_CFC_ (* Continuous Function Chart, elements in execution order *)
#0 <>(SCHU_P2_2_M_MAXSPEED_PE, 0)
#1 AND(SCHU_P2_2_PE_PID_VKL, #0)
#2 Zad_PE:TON(IN: #1, PT: T#2s)
#3 SEL(#2.Q, SCHU_P2_2_M_MAXSPEED_CH, SCHU_P2_2_M_MAXSPEED_PE)
#4 SCHU_P2_2_M_MAXSPEED <= #3
#5 MOVE(EN: NOT #37.Q1, SCHU_P2_2_M_MAXSPEED)
#6 SCHU_P2_2_SPEEDMOTOR <= #5
#7 OR(M1_PUSK, M2_PUSK)
#8 AND(SCHU_P2_2_YA2_M_UST_VKL_UVEL_CHAST, SCHU_P2_2_UE1_TE_NM_UST)
#9 AND(SCHU_P2_2_YA3_M_UST_VKL_UVEL_CHAST, SCHU_P2_2_UE1_TE_NB_UST)
#10 AND(SCHU_P2_2_YA4_M_UST_VKL_UVEL_CHAST, SCHU_P2_2_UE3_TE_B_UST)
#11 AND(#8, #9, #10)
#12 OR(SCHU_P2_2_UE1_TE_M_UST, SCHU_P2_2_UE1_TE_B_UST, SCHU_P2_2_UE3_TE_M_UST, SCHU_P2_2_UST_RE_STOP)
#13 AND(SCHU_P2_2_YA2_B_UST_VKL_STER_REG, SCHU_P2_2_UE1_TE_M_UST)
#14 AND(SCHU_P2_2_UE1_TE_B_UST, SCHU_P2_2_YA3_B_UST_VKL_STER_REG)
#15 AND(SCHU_P2_2_YA4_B_UST_VKL_STER_REG, SCHU_P2_2_UE3_TE_M_UST)
#16 OR(#13, #14, #15)
#17 OR(SCHU_P2_2_M2_OBRBSM, SCHU_P2_2_M1_OBRBSM)
#18 AND(SCHU_P2_2_UST_RE_RABOTA, SCHU_P2_2_AVR_M)
#19 AND(NOT SCHU_P2_2_SA8_DI4_M, SCHU_P2_2_SA1_DI6_M)
#20 OR(SCHU_P2_2_SA1_DO1, SCHU_P2_2_SA8_DO8)
#21 AND(#17, #20)
#22 AND(#11, #21)
#23 SR_START_POV_REG:RS(SET: #22, RESET1: #12)
#24 AND(#16, #21)
#25 AND(#7, #20)
#26 OR(#18, #25)
#27 SEL(#23.Q1, SCHU_P2_2_SPEEDMOTOR, SCHU_P2_2_M_MAXSPEED)
#28 AND(SCHU_P2_2_YA4_M_UST_VKL_STER_REG, SCHU_P2_2_UE3_TE_B_UST)
#29 AND(#23.Q1, #25)
#30 SEL(#29, SCHU_P2_2_M_USKORENIE_PUSK, SCHU_P2_2_M_USKORENIE_UPR)
#31 AND(SCHU_P2_2_UE2_TE_NB_UST, SCHU_P2_2_YA3_M_UST_VKL_STER_REG)
#32 AND(SCHU_P2_2_SA8_DI4_M, NOT SCHU_P2_2_SA1_DI6_M)
#33 AND(SCHU_P2_2_YA2_M_UST_VKL_STER_REG, SCHU_P2_2_UE1_TE_NM_UST)
#34 SEL(SCHU_P2_2_UST_ZIMA, #31, #33)
#35 AND(#28, #34)
#36 OR(SCHU_P2_2_UST_RE_STOP, #35)
#37 SR_START_STER_REG:SR(SET1: #24, RESET: #36)
#38 AND(SCHU_P2_2_M_SB2_STER_REG, NOT #37.Q1)
#39 MOVE(EN: #38, SCHU_P2_2_M_MAXSPEED)
#40 SCHU_P2_2_SPEEDMOTOR <= #39
#41 OR(#23.Q1, #37.Q1)
#42 SEL(#37.Q1, #27, SCHU_P2_2_M_MINSPEED)
#43 SEL(#26, 0, #42)
#44 AND(#25, #37.Q1)
#45 SEL(#44, SCHU_P2_2_M_ZAMEDLENIE_OST, SCHU_P2_2_M_ZAMEDLENIE_UPR)
#46 SEL(SCHU_P2_2_UST_SET_STOP, #45, 1000)
#47 RR:RAMP_REAL(#43, #30, #46, T#1s, -)
#48 MOVE(EN: #41, #47)
#49 SCHU_P2_2_SPEEDMOTOR <= #48
#50 MOVE(EN: SCHU_P2_2_SA1_DO1, #47)
#51 SEL(#50.ENO, 0, #50)
#52 SEL(#19, #51, SCHU_P2_2_M_ZAD_RUCH)
#53 SCHU_P2_2_M1_ZAD_VN <= #52
#54 MOVE(EN: SCHU_P2_2_SA8_DO8, #47)
#55 SEL(#54.ENO, 0, #54)
#56 SEL(#32, #55, SCHU_P2_2_M_ZAD_RUCH)
#57 SCHU_P2_2_M2_ZAD_VN <= #56
#58 RT_KOMVKL_1:R_TRIG(CLK: SCHU_P2_2_UST_RE_PUSK)
#59 MOVE(EN: #58.Q, SCHU_P2_2_M_MAXSPEED)
#60 SCHU_P2_2_SPEEDMOTOR <= #59
#61 RT_KOMVKL_2:R_TRIG(CLK: TRUE)
#62 MOVE(EN: #61.Q, 5)
#63 SCHU_P2_2_M_ZAD_RUCH <= #62
_END_CFC_
END_PROGRAM

(* POU IM/P1_Upr, CFC *)
PROGRAM P1_Upr
VAR
	fb_HVACMS_P1: FB_HVACMotor1Speed;
	SR_P1: SR;
	startDelay_P1: TIME := T#0s;
	stopDelay_P1: TIME := T#0s;
	delayFBC_P1: TIME;
	feedbPT_P1: TIME :=T#10s ;
	delayFBP_P1: TIME := T#10s;
	TON_P1_OTKL_Leto: TON;
	TON_P1_VKL_Leto: TON;
END_VAR
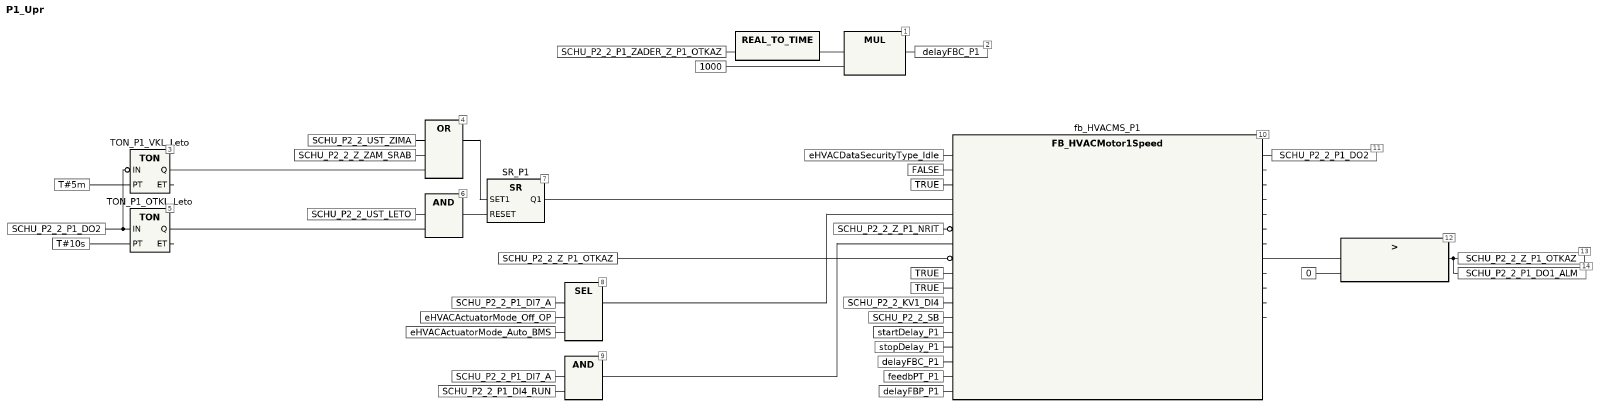
_CFC_ (* Continuous Function Chart, elements in execution order *)
#0 REAL_TO_TIME(SCHU_P2_2_P1_ZADER_Z_P1_OTKAZ)
#1 MUL(#0, 1000)
#2 delayFBC_P1 <= #1
#3 TON_P1_VKL_Leto:TON(IN: NOT SCHU_P2_2_P1_DO2, PT: T#5m)
#4 OR(SCHU_P2_2_UST_ZIMA, SCHU_P2_2_Z_ZAM_SRAB, #3.Q)
#5 TON_P1_OTKL_Leto:TON(IN: SCHU_P2_2_P1_DO2, PT: T#10s)
#6 AND(SCHU_P2_2_UST_LETO, #5.Q)
#7 SR_P1:SR(SET1: #4, RESET: #6)
#8 SEL(SCHU_P2_2_P1_DI7_A, eHVACActuatorMode_Off_OP, eHVACActuatorMode_Auto_BMS)
#9 AND(SCHU_P2_2_P1_DI7_A, SCHU_P2_2_P1_DI4_RUN)
#10 fb_HVACMS_P1:FB_HVACMotor1Speed(eHVACDataSecurityType_Idle, FALSE, TRUE, #7.Q1, #8, NOT SCHU_P2_2_Z_P1_NRIT, #9, NOT SCHU_P2_2_Z_P1_OTKAZ, TRUE, TRUE, SCHU_P2_2_KV1_DI4, SCHU_P2_2_SB, startDelay_P1, stopDelay_P1, delayFBC_P1, feedbPT_P1, delayFBP_P1)
#11 SCHU_P2_2_P1_DO2 <= #10.out 1
#12 >(#10.out 8, 0)
#13 SCHU_P2_2_Z_P1_OTKAZ <= #12
#14 SCHU_P2_2_P1_DO1_ALM <= #12
_END_CFC_
END_PROGRAM

(* POU IM/P2_Upr, CFC *)
PROGRAM P2_Upr
VAR
	fb_HVACMS_P2: FB_HVACMotor1Speed;
	startDelay_P2: TIME := T#0s;
	stopDelay_P2: TIME := T#0s;
	delayFBC_P2: TIME := T#10s;
	feedbPT_P2: TIME :=T#10s ;
	delayFBP_P2: TIME := T#10s;
	errorGeneral: BOOL;
	RS_UE2_SCHU_P2_2_P2_DO3: RS;
	RS_UE3_SCHU_P2_2_P2_DO3: RS;
	UE3_VLmYST: BOOL;
END_VAR
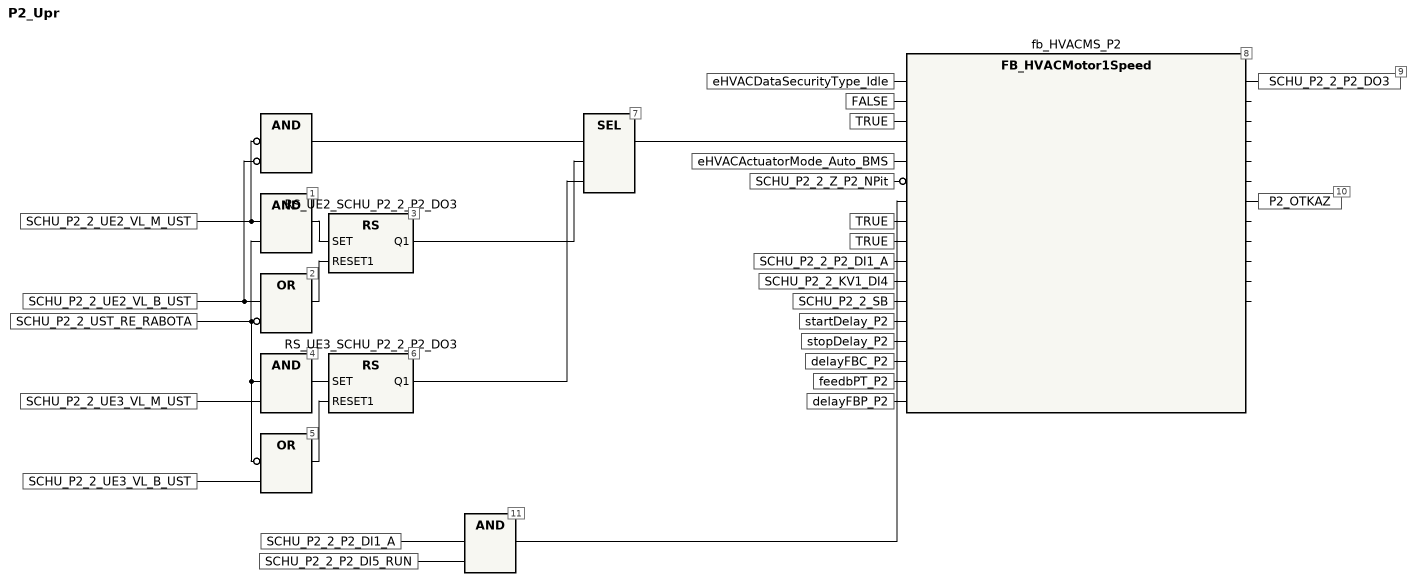
_CFC_ (* Continuous Function Chart, elements in execution order *)
#0 AND(NOT SCHU_P2_2_UE2_VL_M_UST, NOT SCHU_P2_2_UE2_VL_B_UST)
#1 AND(SCHU_P2_2_UE2_VL_M_UST, SCHU_P2_2_UST_RE_RABOTA)
#2 OR(SCHU_P2_2_UE2_VL_B_UST, NOT SCHU_P2_2_UST_RE_RABOTA)
#3 RS_UE2_SCHU_P2_2_P2_DO3:RS(SET: #1, RESET1: #2)
#4 AND(SCHU_P2_2_UST_RE_RABOTA, SCHU_P2_2_UE3_VL_M_UST)
#5 OR(NOT SCHU_P2_2_UST_RE_RABOTA, SCHU_P2_2_UE3_VL_B_UST)
#6 RS_UE3_SCHU_P2_2_P2_DO3:RS(SET: #4, RESET1: #5)
#7 SEL(#0, #3.Q1, #6.Q1)
#8 fb_HVACMS_P2:FB_HVACMotor1Speed(eHVACDataSecurityType_Idle, FALSE, TRUE, #7, eHVACActuatorMode_Auto_BMS, NOT SCHU_P2_2_Z_P2_NPit, #11, TRUE, TRUE, SCHU_P2_2_P2_DI1_A, SCHU_P2_2_KV1_DI4, SCHU_P2_2_SB, startDelay_P2, stopDelay_P2, delayFBC_P2, feedbPT_P2, delayFBP_P2)
#9 SCHU_P2_2_P2_DO3 <= #8.out 1
#10 P2_OTKAZ <= #8.out 7
#11 AND(SCHU_P2_2_P2_DI1_A, SCHU_P2_2_P2_DI5_RUN)
_END_CFC_
END_PROGRAM

(* POU IM/YA1_Upr, CFC *)
PROGRAM YA1_Upr
VAR
	RS_YA1_Open: RS;
	RT_Pusk: R_TRIG;
	RT_OSTANOV: R_TRIG;
	fb_HVACPA: FB_HVAC2PointActuator;

	stokeTime: TIME;
	enableLimitSwitch: BOOL := TRUE;
	FT_PCH_OTKL: R_TRIG;
	TON_PCH_OTKL: TON;
	ZADERJ_SHOD_YA1: TON;
	TON_YA1_Z_ZAM_TE2: TON;
END_VAR
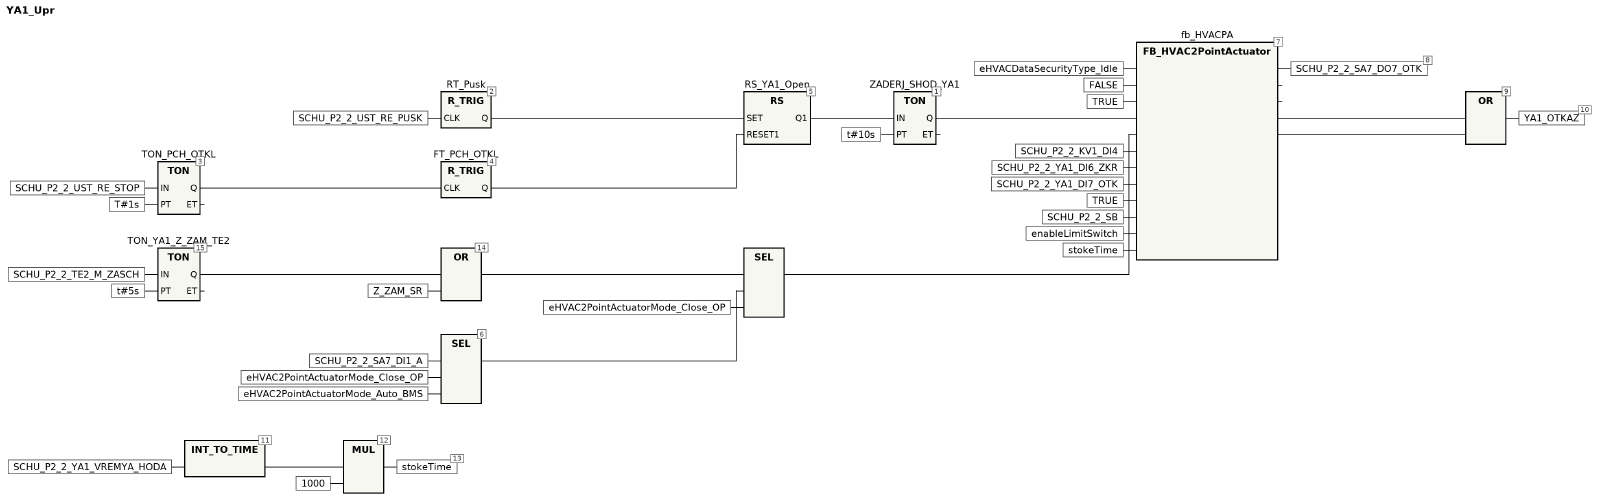
